Fanuc KAREL source: NC0084.KL

-- PROVISIONAL review KL for V770-1; original PC SHA256 de55342cdbaf4e3619bc39b2efbba582919163e6f586774e74815f1eb1a62a43
-- Incomplete behavior may be omitted. Consult companion uncertainty JSON. Do not deploy.
PROGRAM NC0084
%NOLOCKGROUP
-- UNRESOLVED_LOCAL_POOL 2 cells at code offset 3; source declarations unknown
-- DIRECT_LOCAL_WORD_ACCESS alone does not prove INTEGER, REAL, or BOOLEAN
BEGIN
  -- UNRESOLVED_PC offsets 0-8; opcodes 2B,2C,7B
  -- UNRESOLVED_PC offsets 13-20; opcodes 9D,23
  -- UNRESOLVED_PC offsets 25-38; opcodes 21,9D,57,79
  -- UNRESOLVED_PC offsets 43-60; opcodes 21,40,41,42
  -- UNRESOLVED_PC offsets 65-94; opcodes 9D,23,9E,2E,22,7A
  -- UNRESOLVED_PC offsets 99-113; opcodes 21,9D,52,23
  -- UNRESOLVED_PC offsets 118-149; opcodes 20,2C,23,7A,40,41,42
  -- UNRESOLVED_PC offsets 154-178; opcodes 21,2E,52,23,7A,43
  -- UNRESOLVED_PC offsets 183-201; opcodes 21,2E,52,23
  -- UNRESOLVED_PC offsets 211-216; opcodes 7A
  -- UNRESOLVED_PC offsets 221-239; opcodes 21,2E,52,23
  -- UNRESOLVED_PC offsets 249-253; opcodes 7F
  -- UNRESOLVED_PC offsets 258-262; opcodes 27,AA
  -- UNRESOLVED_PC offsets 267-271; opcodes 7F
END NC0084
